Staubli VAL3: MotionCmdVel.pjx

--- MotionCmdVel.pjx ---
Parameters version=s7.8.1 stackSize=5000 millimeterUnit=true
Program file=start.pgx
Program file=stop.pgx
Data file=MotionCmdVel.dtx

--- MotionCmdVel.dtx ---
public num nSequence
public num nVelCmd[6]
public num nCmdType
